(* IEC 61131-3 sources: CodesysTest/export/SX_1195.dev/Plc Logic/Application/IO Handling, 2 files *)

(* ---- universalIOObject.dut.st ---- *)
(*#-#-#-#-#-#-#-#-#-#---Declaration---#-#-#-#-#-#-#-#-#-#-#-#-#*)

TYPE universalIOObject :
STRUCT
	discreteSignal : BOOL;
	signalCommonName : STRING := 'Undefined';
END_STRUCT
END_TYPE

(* ---- Universal_IO_Handler.pou.st ---- *)
(*#-#-#-#-#-#-#-#-#-#---Declaration---#-#-#-#-#-#-#-#-#-#-#-#-#*)

FUNCTION_BLOCK Universal_IO_Handler
VAR_INPUT
	initSignal: universalIOObject;
END_VAR
VAR_IN_OUT
	mappedSignal:BOOL;
END_VAR(*#-#-#-#-#-#-#-#-#-#---Implementation---#-#-#-#-#-#-#-#-#-#-#-#-#*)

mappedSignal:=initSignal.discreteSignal;
